// TIA Portal V16 export
// export: Created 2022-02-28T20:45:46.302721Z, ExportSetting WithDefaults, DisplayName Totally Integrated Automation Portal, DisplayVersion V16, DisplayName TIA Portal Version Control Interface, DisplayVersion V16, DisplayName TIA Portal Openness, DisplayVersion V16, DisplayName STEP 7 Professional, DisplayVersion V16, DisplayName STEP 7 Safety, DisplayVersion V16, DisplayName WinCC Advanced, DisplayVersion V16
DATA_BLOCK "05_General"   // DB5
{ S7_Optimized_Access := 'TRUE' }
VERSION : 0.1
// stored: AutoNumber true, DBAccessibleFromOPCUA true, IsOnlyStoredInLoadMemory false, IsRetainMemResEnabled false, IsWriteProtectedInAS false, MemoryReserve 100
   VAR
      MP_Perifericos_Ok : Bool;   // Confirmación perifericos pistilos
      "MP_Habilita_Start-Stop" : Bool;   // Habilitar Remoto pistilos
      MP_Start_HMI : Bool;   // Start Remoto Pistilos
      MP_Stop_HMI : Bool;   // Stop Remoto Pistilos
      MPF_Perifericos_OK : Bool;   // Confirmación perifericos pentoflex
      "MPF_Habilita_Start-Stop" : Bool;   // Habilitar Remoto pentoflex
      MPF_Start_HMI : Bool;   // Start Remoto Pentoflex
      MP_Stop_HMI_1 : Bool;   // Stop Remoto Pentoflex
   END_VAR
BEGIN
END_DATA_BLOCK
